% RSLogix 500 project P9_IVANOVSKI_M.RSS, saved by version 8.30.00.16 %
PROJECT "UNTITLED"    % processor: Bul.1763 MicroLogix 1100 Series B %

PROGRAM FILES
  LAD 2 "MAIN"  3 rungs
  LAD 3 "IO"  5 rungs
  LAD 4 "CONTROLS"  3 rungs

DATA FILES
  O0 OUTPUT  4 elements
  I1 INPUT  6 elements
  S2 STATUS  66 elements
  B3 BINARY  2 elements
  T4 TIMER  1 elements
  C5 COUNTER  1 elements
  R6 CONTROL  1 elements
  N7 INTEGER  4 elements
  F8 FLOAT  1 elements
  ST9 STRING  15 elements

LADDER 2 "MAIN"
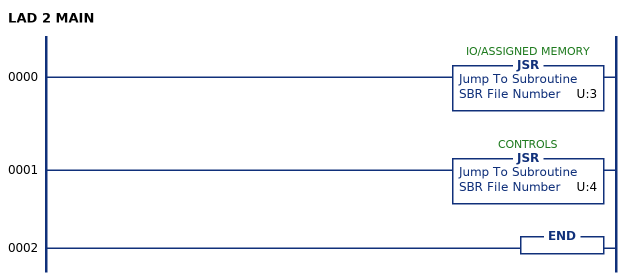
% Rung: 0 %
SOR JSR U:3 EOR
%   U:3  "IO/ASSIGNED MEMORY" %
% Rung: 1 %
SOR JSR U:4 EOR
%   U:4  "CONTROLS" %
% Rung: 2 %
SOR END EOR

LADDER 3 "IO"
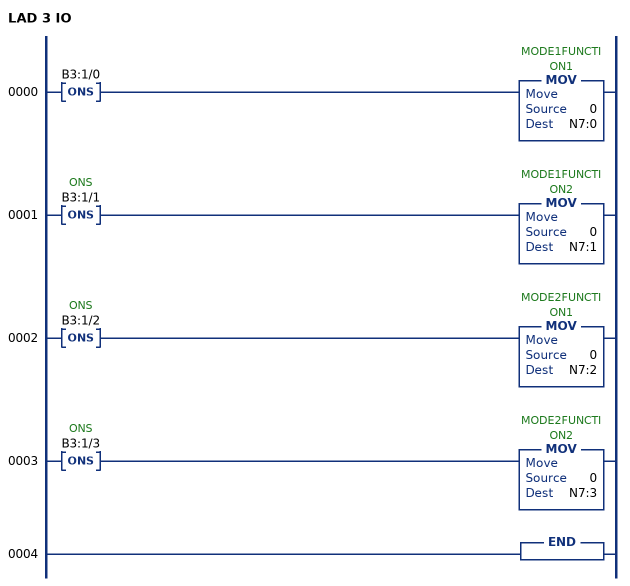
% Rung: 0 %
SOR ONS B3:1/0 MOV 0 N7:0 EOR
%   N7:0  "MODE1FUNCTION1" %
% Rung: 1 %
SOR ONS B3:1/1 MOV 0 N7:1 EOR
%   B3:1/1  "ONS" %
%   N7:1  "MODE1FUNCTION2" %
% Rung: 2 %
SOR ONS B3:1/2 MOV 0 N7:2 EOR
%   B3:1/2  "ONS" %
%   N7:2  "MODE2FUNCTION1" %
% Rung: 3 %
SOR ONS B3:1/3 MOV 0 N7:3 EOR
%   B3:1/3  "ONS" %
%   N7:3  "MODE2FUNCTION2" %
% Rung: 4 %
SOR END EOR

LADDER 4 "CONTROLS"
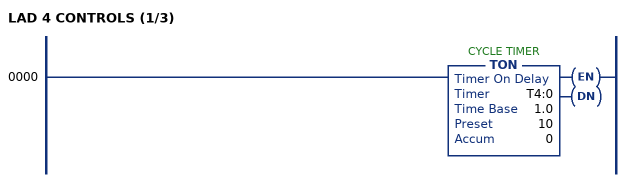
% Rung: 0 %
SOR TON T4:0 1.0 10 0 EOR
%   T4:0  "CYCLE TIMER" %

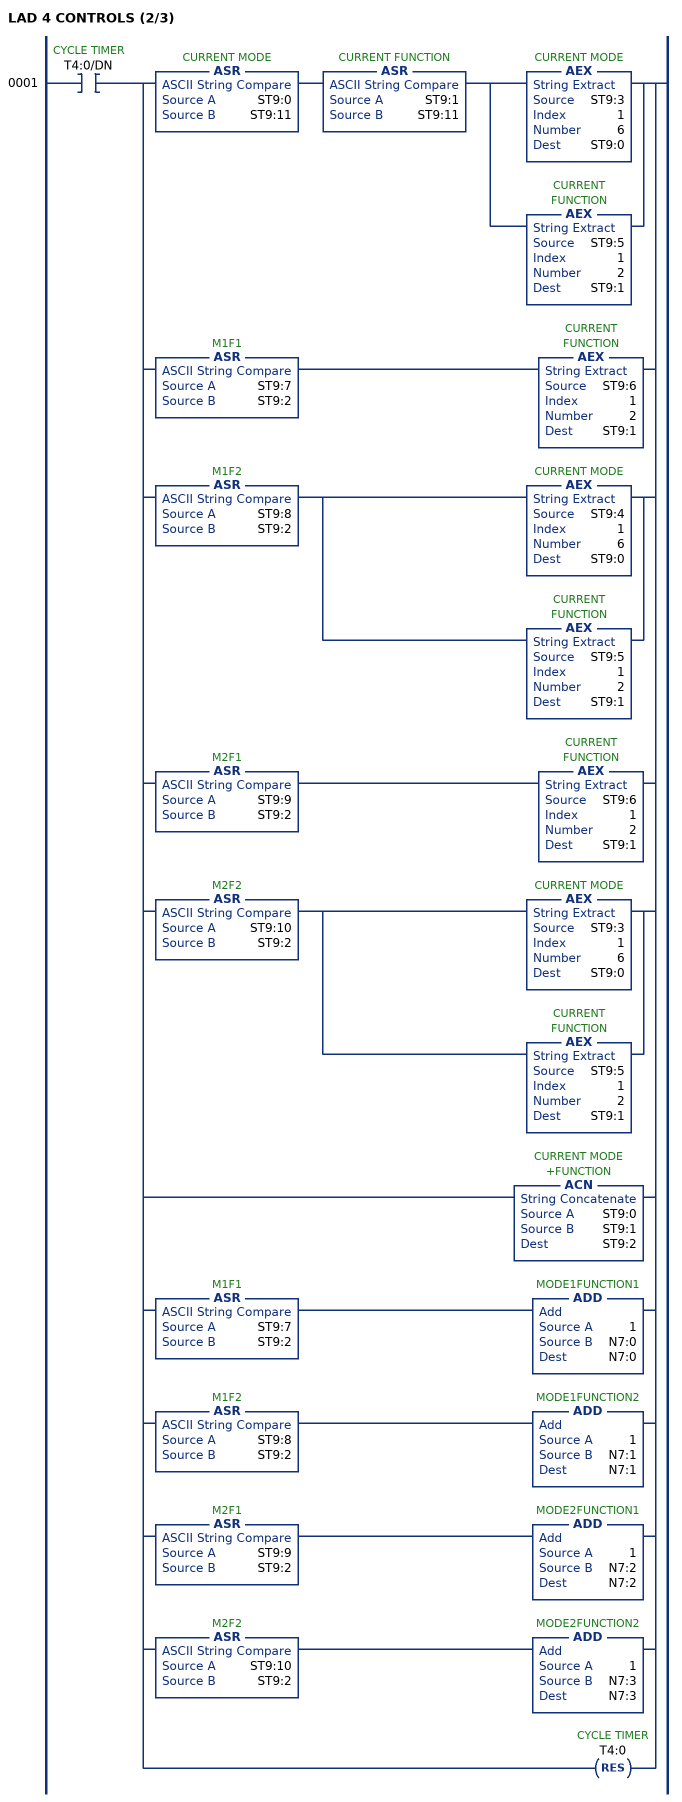
% Rung: 1 %
SOR XIC T4:0/DN BST ASR ST9:0 ST9:11 ASR ST9:1 ST9:11 BST AEX ST9:3 1 6 ST9:0 NXB AEX ST9:5 1 2 ST9:1 BND NXB ASR ST9:7 ST9:2 AEX ST9:6 1 2 ST9:1 NXB ASR ST9:8 ST9:2 BST AEX ST9:4 1 6 ST9:0 NXB AEX ST9:5 1 2 ST9:1 BND NXB ASR ST9:9 ST9:2 AEX ST9:6 1 2 ST9:1 NXB ASR ST9:10 ST9:2 BST AEX ST9:3 1 6 ST9:0 NXB AEX ST9:5 1 2 ST9:1 BND NXB ACN ST9:0 ST9:1 ST9:2 NXB ASR ST9:7 ST9:2 ADD 1 N7:0 N7:0 NXB ASR ST9:8 ST9:2 ADD 1 N7:1 N7:1 NXB ASR ST9:9 ST9:2 ADD 1 N7:2 N7:2 NXB ASR ST9:10 ST9:2 ADD 1 N7:3 N7:3 NXB RES T4:0 BND EOR
%   T4:0  "CYCLE TIMER" %
%   ST9:0  "CURRENT MODE" %
%   ST9:1  "CURRENT FUNCTION" %
%   ST9:3  "MODE 1" %
%   ST9:5  "FUNCTION 1" %
%   ST9:7  "M1F1" %
%   ST9:2  "CURRENT MODE +FUNCTION" %
%   ST9:6  "FUNCTION 2" %
%   ST9:8  "M1F2" %
%   ST9:4  "MODE 2" %
%   ST9:9  "M2F1" %
%   ST9:10  "M2F2" %
%   N7:0  "MODE1FUNCTION1" %
%   N7:1  "MODE1FUNCTION2" %
%   N7:2  "MODE2FUNCTION1" %
%   N7:3  "MODE2FUNCTION2" %

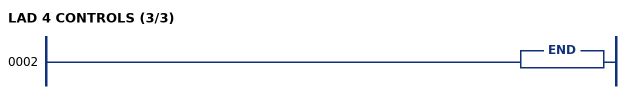
% Rung: 2 %
SOR END EOR

OTHER DOCUMENTED ADDRESSES
  B3:1/4  "ONS"

DATA TABLE (non-zero values as saved)
DATA T4
% .PRE .ACC %
% T4:0 % 10 0
DATA ST9
% ST9:3 % "MODE-1"
% ST9:4 % "MODE-2"
% ST9:5 % "F1"
% ST9:6 % "F2"
% ST9:7 % "MODE-1F1"
% ST9:8 % "MODE-1F2"
% ST9:9 % "MODE-2F1"
% ST9:10 % "MODE-2F2"
